// Writes a string field value, without a tag, to the stream. The data is length-prefixed.
FUNCTION F_WriteString : HRESULT
VAR_INPUT
    stBuffer    : ST_Span;
END_VAR
VAR_IN_OUT
    stState     : ST_WriterInternalState;
END_VAR
VAR_IN_OUT CONSTANT
    sValue  : T_ProtobufMaxString;
END_VAR
VAR
    tAnyString : T_AnyString;
END_VAR

F_WriteString := S_OK;

tAnyString.pValue := ADR(sValue[0]);
tAnyString.TypeClass := __SYSTEM.TYPE_CLASS.TYPE_STRING;
tAnyString.diSize := SIZEOF(T_ProtobufMaxString);

F_WriteString := F_WriteRawString(stBuffer, stState, tAnyString);

END_FUNCTION

(* stored: Version 1.1.0.1
   POU F_WriteString: Id {09fd94e5-4952-4576-a108-1cdf6abd18f4}, SpecialFunc None *)
